Universal Robots URScript: 20240827vision.script

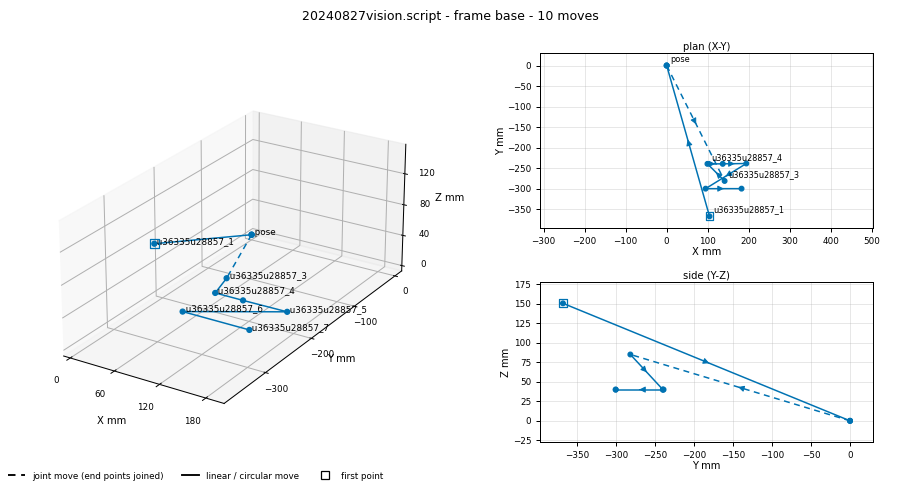
[picture p0: tool path of 20240827vision.script in frame base, 10 of 11 moves have a stored position in this frame; points joined in program order, loops and branches not executed]
def P20240827vision():
  global _hidden_verificationVariable=0
  set_safety_mode_transition_hardness(0)
  set_target_payload(1.500000, [0.001000, -0.003000, 0.050000], [0.003026, 0.003026, 0.003026, 0.000000, 0.000000, 0.000000])
  set_gravity([0.0, 0.0, 9.82])
  set_tcp(p[-1.7E-4,0.0,0.19294999999999998,0.0,0.0,0.0])
  set_standard_analog_input_domain(0, 1)
  set_standard_analog_input_domain(1, 1)
  set_tool_analog_input_domain(0, 1)
  set_tool_analog_input_domain(1, 1)
  set_analog_outputdomain(0, 1)
  set_analog_outputdomain(1, 0)
  set_input_actions_to_default()
  set_tool_digital_input_action(0, "freedrive")
  set_tool_communication(True, 115200, 0, 1, 1.5, 3.5)
  set_tool_output_mode(0)
  set_tool_digital_output_mode(0, 1)
  set_tool_digital_output_mode(1, 1)
  set_tool_voltage(24)
  global i_var_1=p[0.31, 0, 0, 0, 0, 0]
  global u24179u38754_1=p[0.0,0.0,0.0,0.0,0.0,0.0]
  global u24179u38754_2=p[0.2,0.6,0.4,-1.4839444017850547,-0.07419722008925289,-2.225916602677581]
  global u24179u38754_3=p[0.1459477485431481,-0.10308445883660293,0.13857682671027435,-0.008977024873201634,0.014216906208388691,-2.4400986907073663]
  global u28857_1=p[0.10203918836050063,-0.5259531579406657,0.376430278847906,-0.18768520041296463,-3.1325095402283982,-0.09669790600413578]
  global u28857_2=p[0.0665007526844362,-0.3872123180436422,0.638459113340625,-0.320095108678139,-2.6903368475934015,1.4700117755369673]
  global u30452u32447_1=p[0.0,0.0,0.0,0.0,0.0,0.0]
  step_count_1a284065_73db_4a87_86ac_5485ac17be38 = 0.0
  thread Step_Counter_Thread_03664bf6_442c_4511_b66b_bd81e107a8a9():
    while (True):
      step_count_1a284065_73db_4a87_86ac_5485ac17be38 = step_count_1a284065_73db_4a87_86ac_5485ac17be38 + 1.0
      sync()
    end
  end
  run Step_Counter_Thread_03664bf6_442c_4511_b66b_bd81e107a8a9()
  global u36335u28857_1_p=p[.104511126124, -.367886971260, .150559642288, -1.949339747521, -1.826249279458, -.604804033827]
  global u36335u28857_1_q=[1.491742491722107, -1.4001733523658295, 1.7467568556415003, -1.3199103635600586, -1.573672119771139, 1.5610108375549316]
  global u36335u28857_3_p=p[.141277002130, -.281524029863, .085000000000, 2.221117452349, 2.221081034482, .002926406814]
  global u36335u28857_3_q=[1.5945374000737473, -1.9677764116104068, 2.4363131384382193, -2.0391606082839537, -1.569434457309896, 1.5968019570169858]
  global u36335u28857_4_p=p[.099451506469, -.239827777747, .040000000000, 2.221375407522, 2.221468721165, -.000030434756]
  global u36335u28857_4_q=[1.4215074140541617, -2.1065920354457894, 2.628929087112269, -2.0939256438267098, -1.5711927999278963, 1.4234675481607901]
  global u36335u28857_2_p=p[.136756227030, -.239835520679, .040000000000, 2.221364653615, 2.221479599810, -.000043033614]
  global u36335u28857_2_q=[1.582221072329581, -2.030634877917432, 2.5989922896895443, -2.1399526785968703, -1.5712859869972782, 1.584240456074161]
  global u36335u28857_5_p=p[.194273191653, -.238974860860, .040000000000, 2.221394498094, 2.221487650310, -.000001601352]
  global u36335u28857_5_q=[1.8031859177960374, -1.9022351259993915, 2.5356426673992996, -2.204964891086526, -1.5714183059403517, 1.805335628500325]
  global u36335u28857_6_p=p[.094922978788, -.300331282322, .040000000000, 2.221451764059, 2.221386493456, -.000099951617]
  global u36335u28857_6_q=[1.4371962570780292, -1.8769673279171206, 2.521101597790169, -2.2157602880765346, -1.571456264094719, 1.4394418991969617]
  global u36335u28857_7_p=p[.182597025114, -.300301124632, .040000000000, -2.221435645453, -2.221373284537, .000001847065]
  global u36335u28857_7_q=[1.7256884767632812, -1.7564912882892294, 2.441004347935132, -2.256027493222483, -1.5715866918052939, 1.7280571366920494]
  while (True):
    $ 2 "机器人程序"
    $ 3 "MoveJ"
    $ 4 "路点_1" "breakAfter"
    movej(u36335u28857_1_q, a=1.3962634015954636, v=1.0471975511965976)
    $ 5 "move = rpc_factory('xmlrpc','http://192.168.1.5:9121/RPC2')"
    move = rpc_factory("xmlrpc","http://192.168.1.5:9121/RPC2")
    $ 6 "usb = rpc_factory('xmlrpc','http://192.168.1.2:9120/RPC2')"
    usb = rpc_factory("xmlrpc","http://192.168.1.2:9120/RPC2")
    $ 7 "usb.open()"
    usb.open()
    $ 11 "n≔0"
    global n=0
    $ 12 "循环"
    while (True):
      $ 13 "MoveJ"
      $ 14 "路点_1" "breakAfter"
      movej(get_inverse_kin(u36335u28857_1_p, qnear=u36335u28857_1_q), a=1.3962634015954636, v=1.5707963267948966)
      $ 15 "n≔n + 1"
      global n=n + 1
      $ 16 "move.take_photo()"
      move.take_photo()
      $ 17 "弹出窗口: 123"
      popup("123", "消息", False, False, blocking=True)
      $ 18 "循环 5 次数"
      u24490u29615_2 = 0
      while (u24490u29615_2 < 5):
        $ 20 "obj_num≔n"
        global obj_num=n
        $ 22 "pose≔p[0.0,0.0,0.0,2.221,2.221,0.004]"
        global pose=p[0.0,0.0,0.0,2.221,2.221,0.004]
        $ 24 "var_2≔move.move_pose(obj_num)"
        global var_2=move.move_pose(obj_num)
        $ 26 "pose[0]=var_2[0]"
        pose[0]=var_2[0]
        $ 27 "pose[1]=var_2[1]"
        pose[1]=var_2[1]
        $ 28 "pose[2]=0.1"
        pose[2]=0.1
        $ 29 "MoveL"
        $ 30 "pose" "breakAfter"
        movel(pose, a=0.15, v=0.4)
        $ 31 "pose[2]=0.003"
        pose[2]=0.003
        $ 32 "MoveL"
        $ 33 "pose" "breakAfter"
        movel(pose, a=0.15, v=0.4)
        $ 34 "usb.adaptiveClose()"
        usb.adaptiveClose()
        $ 35 "pose[2]=0.1"
        pose[2]=0.1
        $ 36 "MoveL"
        $ 37 "pose" "breakAfter"
        movel(pose, a=0.25, v=1.5)
        $ 38 "MoveJ"
        $ 39 "路点_3" "breakAfter"
        movej(get_inverse_kin(u36335u28857_3_p, qnear=u36335u28857_3_q), a=1.3962634015954636, v=1.7453292519943295)
        $ 40 "If n==1"
        if (n==1):
          $ 41 "MoveL"
          $ 42 "路点_4" "breakAfter"
          movel(u36335u28857_4_p, a=0.15, v=0.4)
        end
        $ 43 "If n==2"
        if (n==2):
          $ 44 "MoveL"
          $ 45 "路点_2" "breakAfter"
          movel(u36335u28857_2_p, a=0.15, v=0.4)
        end
        $ 46 "If n==3"
        if (n==3):
          $ 47 "MoveL"
          $ 48 "路点_5" "breakAfter"
          movel(u36335u28857_5_p, a=0.15, v=0.4)
        end
        $ 49 "If n==4"
        if (n==4):
          $ 50 "MoveL"
          $ 51 "路点_6" "breakAfter"
          movel(u36335u28857_6_p, a=0.15, v=0.4)
        end
        $ 52 "If n==5"
        if (n==5):
          $ 53 "MoveL"
          $ 54 "路点_7" "breakAfter"
          movel(u36335u28857_7_p, a=0.15, v=0.4)
        end
        $ 55 "n=n+1"
        n=n+1
        $ 56 "usb.open()"
        usb.open()
        u24490u29615_2 = u24490u29615_2 + 1
      end
    end
  end
end
